SUBAPPLICATION GreenBlueBackground1_AXS (* Hintergrundfarbe (TRUE -> Blau, FALSE -> Weiß) für 1 Objekt (AX-Adapter) *)
  (* Standard: 61499-2; Description: Copyright (c) 2022 HR Agrartechnik GmbH This program and the accompanying materials are made available under the terms of the Eclipse Public License 2.0 which is available at https://www.eclipse.org/legal/epl-2.0/ SPDX-License-Identifier: EPL-2.0 *)
  (* Version 1.0, 2022-11-10, Franz Höpfinger, HR Agrartechnik GmbH *)
  PACKAGE MyLib::sys;
  IMPORT isobus::UT::Q::const::IDs::ID_NULL;
  IMPORT isobus::UT::Q::const::colours::COLOR_BLUE;
  IMPORT isobus::UT::Q::const::colours::COLOR_WHITE;
  IMPORT isobus::UT::Q::types::s1ObjectID;
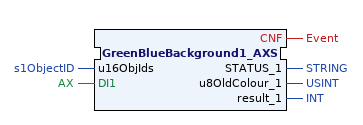
  EVENT_OUTPUT
    CNF; (* Execution Confirmation *)
  END_EVENT
  VAR_INPUT
    u16ObjIds : isobus::UT::Q::types::s1ObjectID := (u16ObjId := ID_NULL); (* Object ID *)
  END_VAR
  VAR_OUTPUT
    STATUS_1 : STRING; (* Service Status *)
    u8OldColour_1 : USINT; (* Old value of ID *)
    result_1 : INT; (* retval see description *)
  END_VAR
  SOCKETS
    DI1 : adapter::types::unidirectional::AX; (* Selector *)
  END_SOCKETS
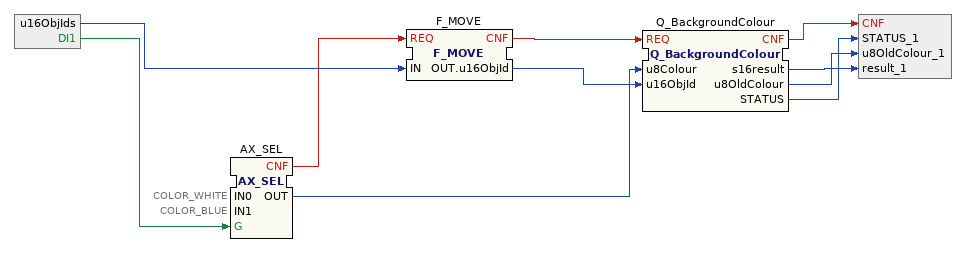
  FBS
    Q_BackgroundColour : isobus::UT::Q::Q_BackgroundColour;
    AX_SEL : adapter::iec61131::selection::AX_SEL(IN0 := COLOR_WHITE, IN1 := COLOR_BLUE);
    F_MOVE : iec61131::selection::F_MOVE; {SET_ATTRIBUTE(DataType, isobus::UT::Q::types::s1ObjectID)}
  END_FBS
  EVENT_CONNECTIONS
    Q_BackgroundColour.CNF TO CNF;
    F_MOVE.CNF TO Q_BackgroundColour.REQ;
    AX_SEL.CNF TO F_MOVE.REQ;
  END_CONNECTIONS
  DATA_CONNECTIONS
    Q_BackgroundColour.s16result TO result_1;
    Q_BackgroundColour.u8OldColour TO u8OldColour_1;
    Q_BackgroundColour.STATUS TO STATUS_1;
    AX_SEL.OUT TO Q_BackgroundColour.u8Colour;
    u16ObjIds TO F_MOVE.IN;
    F_MOVE.OUT.u16ObjId TO Q_BackgroundColour.u16ObjId;
  END_CONNECTIONS
  ADAPTER_CONNECTIONS
    DI1 TO AX_SEL.G;
  END_CONNECTIONS
END_SUBAPPLICATION
